PROGRAM MAIN
VAR
END_VAR


// Main Routine
Initialize();
MainCycle();
FaultDetection();
Counters();
HMIUpdates();

//LogicTester();
LogicTester2();

END_PROGRAM

(* stored: Version 1.1.0.1
   POU MAIN: Id {527f438a-01c8-4e6e-8aa4-aea9433d8d02}, SpecialFunc None *)
